# EPICS IOC start-up script: test/startup/st.sim-indexer.iocsh
epicsEnvSet("MOTOR_PORT",      "$(SM_MOTOR_PORT=MCU1)")

epicsEnvSet("IPADDR",          "$(SM_IPADDR=127.0.0.1)")
epicsEnvSet("IPPORT",          "$(SM_IPPORT=48898)")
epicsEnvSet("AMSNETIDIOC",     "$(SM_AMSNETID=127.0.0.1.1.1)")
epicsEnvSet("ASYN_PORT",       "$(SM_ASYN_PORT=MC_CPU1)")
epicsEnvSet("P",               "$(SM_P=IOC:)")
epicsEnvSet("R",               "")
epicsEnvSet("PREC",            "$(SM_PREC=3)")
# 6 axes: 4 motors, axis 5 is shutter, 6 is pneumatic, 7 is carousel, 8 is analog output
epicsEnvSet("ECM_NUMAXES",     "8")
epicsEnvSet("ADSPORT",         "$(ECM_ADSPORT=852)")
epicsEnvSet("ECM_OPTIONS",     "adsPort=$(ADSPORT);amsNetIdRemote=127.0.0.1.1.1;amsNetIdLocal=$(AMSNETIDIOC)"

# Do not start the poller yet
epicsEnvSet("ECM_MOVINGPOLLPERIOD", "0")
epicsEnvSet("ECM_IDLEPOLLPERIOD", "0")
< ethercatmcController.iocsh

#
# Cabinet status
#
epicsEnvSet("AXIS_NO",         "0")
epicsEnvSet("R",               "Cabinet")
epicsEnvSet("DESC",            "Cabinet")
epicsEnvSet("EGU",             "Cabinet")
< ethercatmcCabinet.iocsh

#
# Axis 1
#
epicsEnvSet("AXISCONFIG",      "")
epicsEnvSet("R",               "$(SM_R=m1)")
epicsEnvSet("AXIS_NO",         "$(SM_AXIS_NO=1)")
epicsEnvSet("RAWENCSTEP_ADEL", 0)
epicsEnvSet("RAWENCSTEP_MDEL", 0)
< ethercatmcIndexerAxis.iocsh
< ethercatmcAxisdebug.iocsh
< ethercatmcOpenClutch.iocsh
# Test records
< ethercatmcTestInputRecordAlarm.iocsh
# Aux bits as bi records;
# R:Record name
# P: asynParam name
epicsEnvSet("AUX_BIT_NAME_R",  "notHomed")
epicsEnvSet("AUX_BIT_NAME_P",  "AUXBITnotHomed")
< ethercatmcAuxBitAsBiRecord.iocsh

# Predefined Positions
# NVL: Input Value Location (INLINK)
epicsEnvSet("NVL",             "")
epicsEnvSet("EGU",             "")
< ethercatmcDefPos.iocsh

#
# Axis 2
#
epicsEnvSet("AXISCONFIG",      "")
epicsEnvSet("R",               "$(SM_R=m2)")
epicsEnvSet("AXIS_NO",         "$(SM_AXIS_NO=2)")
epicsEnvSet("RAWENCSTEP_ADEL", 0)
epicsEnvSet("RAWENCSTEP_MDEL", 0)
< ethercatmcIndexerAxis.iocsh
< ethercatmcAxisdebug.iocsh
#< ethercatmcOpenClutch.iocsh

#
# Axis 3
#
epicsEnvSet("AXISCONFIG",      "")
epicsEnvSet("R",               "$(SM_R=m3)")
epicsEnvSet("AXIS_NO",         "$(SM_AXIS_NO=3)")
epicsEnvSet("RAWENCSTEP_ADEL", 0)
epicsEnvSet("RAWENCSTEP_MDEL", 0)
< ethercatmcIndexerAxis.iocsh
< ethercatmcAxisdebug.iocsh
#< ethercatmcOpenClutch.iocsh

#
# Axis 4
#
epicsEnvSet("AXISCONFIG",      "")
epicsEnvSet("R",               "$(SM_R=m4)")
epicsEnvSet("AXIS_NO",         "$(SM_AXIS_NO=4)")
epicsEnvSet("RAWENCSTEP_ADEL", 0)
epicsEnvSet("RAWENCSTEP_MDEL", 0)
< ethercatmcIndexerAxis.iocsh
< ethercatmcAxisdebug.iocsh
#< ethercatmcOpenClutch.iocsh

#
# Axis 5, shutter
#
epicsEnvSet("AXISCONFIG",      "")
epicsEnvSet("R",               "Sht")
epicsEnvSet("AXIS_NO",         "5")
< ethercatmcShutter.iocsh

# Motorrecord to debug
#epicsEnvSet("R",    "Shutter")
#< ethercatmcIndexerAxis.iocsh

#
# Axis 6, pneumatic with ErrId
#
epicsEnvSet("AXISCONFIG",      "")
epicsEnvSet("R",               "Pneu")
epicsEnvSet("AXIS_NO",         "6")
< ethercatmcShutter.iocsh
# Motorrecord and debug needed for the automatic tests/943
< ethercatmcIndexerAxis.iocsh
< ethercatmcAxisdebug.iocsh

#
# Axis 7, carousel with ErrId
#
epicsEnvSet("AXISCONFIG",      "")
epicsEnvSet("R",               "Carousel")
epicsEnvSet("AXIS_NO",         "7")
# Motorrecord and debug needed for the automatic tests/943
< ethercatmcIndexerAxis.iocsh
< ethercatmcAxisdebug.iocsh

#
# CHNO 1: analog output with readback.
#
epicsEnvSet("AXISCONFIG",      "")
epicsEnvSet("R",               "AnalogOutput")
epicsEnvSet("CHNO",            "1")
epicsEnvSet("ASYNPARAMNAME",   "ANALOGOUTPUT")
epicsEnvSet("PREC",            "3")
epicsEnvSet("DESC",            "AnalogOutput")
epicsEnvSet("EGU",             "mm")
< ethercatmcAnalogOutputReadback.iocsh

# Faster polling
epicsEnvSet("MOVINGPOLLPERIOD",  "100")
epicsEnvSet("IDLEPOLLPERIOD",    "100")
ethercatmcStartPoller("$(MOTOR_PORT)", "$(MOVINGPOLLPERIOD)", "$(IDLEPOLLPERIOD)")
